TYPE ST_System_FBT_Steuerung :
STRUCT
	Freigabe			: ST_Steuerung_auto_manu_BOOL;
	Freigabe_Deakt		: ST_Steuerung_auto_manu_BOOL;
	Betrieb_Anford		: ST_Steuerung_auto_manu_opti_BOOL;

	Regelung_Modus		: ST_Steuerung_auto_manu_opti_SINT;
	Regelung_Nachtabs	: ST_Steuerung_auto_manu_opti_BOOL;
	Regelung_Sollw		: ST_Steuerung_auto_manu_opti_REAL;

	Test2 : REAL;

	Quittierung			: BOOL;
END_STRUCT
END_TYPE

(* stored: Version 1.1.0.1, ProductVersion 3.1.4024.9
   DUT ST_System_FBT_Steuerung: Id {becaafa2-19b9-4ad5-9bc6-c7ef3abda682} *)
